Omron CX-Programmer project NewProject (CX-Programmer 9.73)

# PLC bagagli: CPM1(CPM1A) CPU20

## Global symbols (name address type ; comment)
0.01 BOOL  ; EntryBalance1
0.02 BOOL  ; SensorBalance2
0.03 BOOL  ; SensorBalance3
0.04 BOOL  ; WeightC1
0.05 BOOL  ; XRayC1
0.06 BOOL  ; WeightC2
0.07 BOOL  ; XRayC2
0.08 BOOL  ; WeightC3
0.09 BOOL  ; Tag3
0.10 BOOL  ; Tag
0.11 BOOL  ; SensorEntryRoll1
0.12 BOOL  ; SensorRoll2
0.13 BOOL  ; SensorRoll3
0.14 BOOL  ; SensorRoll2
0.15 BOOL  ; SensorRoll3
10.00 BOOL  ; BagOnBalance1
10.01 BOOL  ; Position Control1
10.02 BOOL  ; Position Control2
10.03 BOOL  ; Position Control3
10.04 BOOL  ; RemLW1
10.05 BOOL  ; RemLW2
10.06 BOOL  ; RemLW3
10.07 BOOL  ; Container brought to destination
10.08 BOOL  ; Roll3
10.09 BOOL  ; Roll2
10.10 BOOL  ; Roll1
10.11 BOOL  ; Roll1
10.12 BOOL  ; Roll2
10.13 BOOL  ; Roll3
10.14 BOOL  ; FlagCont
11.01 BOOL  ; Roll1
11.02 BOOL  ; Roll2
11.03 BOOL  ; Roll3
1.01 BOOL  ; EntryL1
1.02 BOOL  ; ExitL1
1.03 BOOL  ; EntryL2
1.04 BOOL  ; ExitL2
1.05 BOOL  ; EntryL3
1.06 BOOL  ; ExitL3
1.07 BOOL  ; Tag1
1.08 BOOL  ; Tag2
1.09 BOOL  ; Tag3
1.10 BOOL  ; Exit2Full
1.11 BOOL  ; EndRoll2
1.12 BOOL  ; ExitSensorRoll1
1.13 BOOL  ; SensorRoll3
1.14 BOOL  ; SensorRoll1
1.15 BOOL  ; SensorRoll2
CNT127 BOOL  ; ContainerL
HR0.01 BOOL  ; test1
HR0.04 BOOL  ; test1
TIM000 BOOL  ; 10s to change container

## Program NewProgram1 (no task)
Local symbols
SensorRoll2 1.15 BOOL  ; SensorRoll2
XRayC1 BOOL

### Section Section1

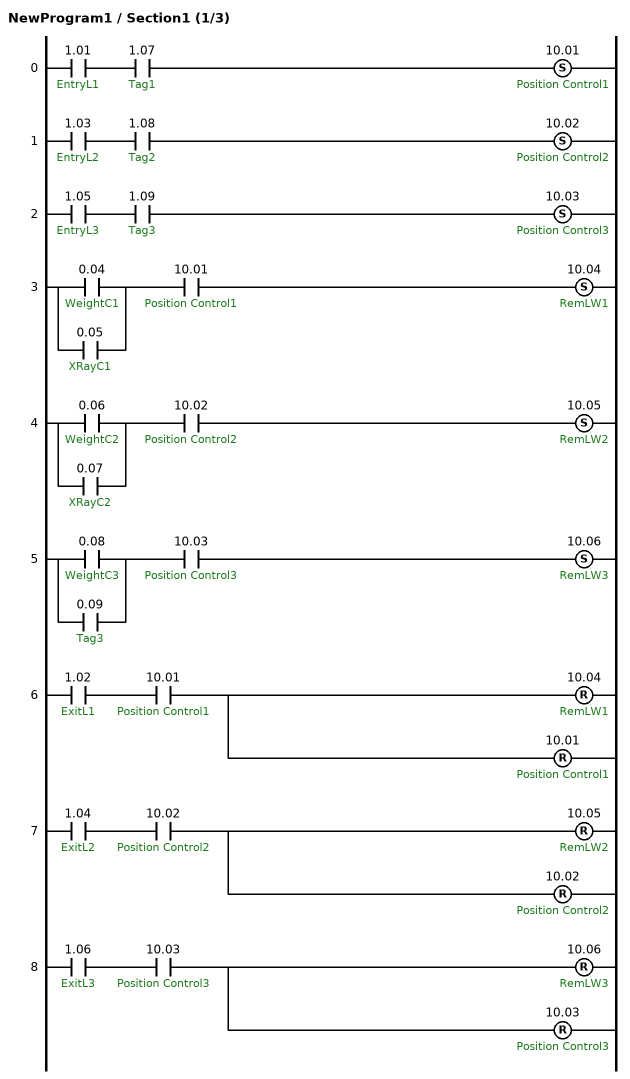
; rung 0
LD 1.01  ; EntryL1
AND 1.07  ; Tag1
SET 10.01  ; Position Control1
; rung 1
LD 1.03  ; EntryL2
AND 1.08  ; Tag2
SET 10.02  ; Position Control2
; rung 2
LD 1.05  ; EntryL3
AND 1.09  ; Tag3
SET 10.03  ; Position Control3
; rung 3
LD 0.04  ; WeightC1
OR 0.05  ; XRayC1
AND 10.01  ; Position Control1
SET 10.04  ; RemLW1
; rung 4
LD 0.06  ; WeightC2
OR 0.07  ; XRayC2
AND 10.02  ; Position Control2
SET 10.05  ; RemLW2
; rung 5
LD 0.08  ; WeightC3
OR 0.09  ; Tag3
AND 10.03  ; Position Control3
SET 10.06  ; RemLW3
; rung 6
LD 1.02  ; ExitL1
AND 10.01  ; Position Control1
RSET 10.04  ; RemLW1
RSET 10.01  ; Position Control1
; rung 7
LD 1.04  ; ExitL2
AND 10.02  ; Position Control2
RSET 10.05  ; RemLW2
RSET 10.02  ; Position Control2
; rung 8
LD 1.06  ; ExitL3
AND 10.03  ; Position Control3
RSET 10.06  ; RemLW3
RSET 10.03  ; Position Control3

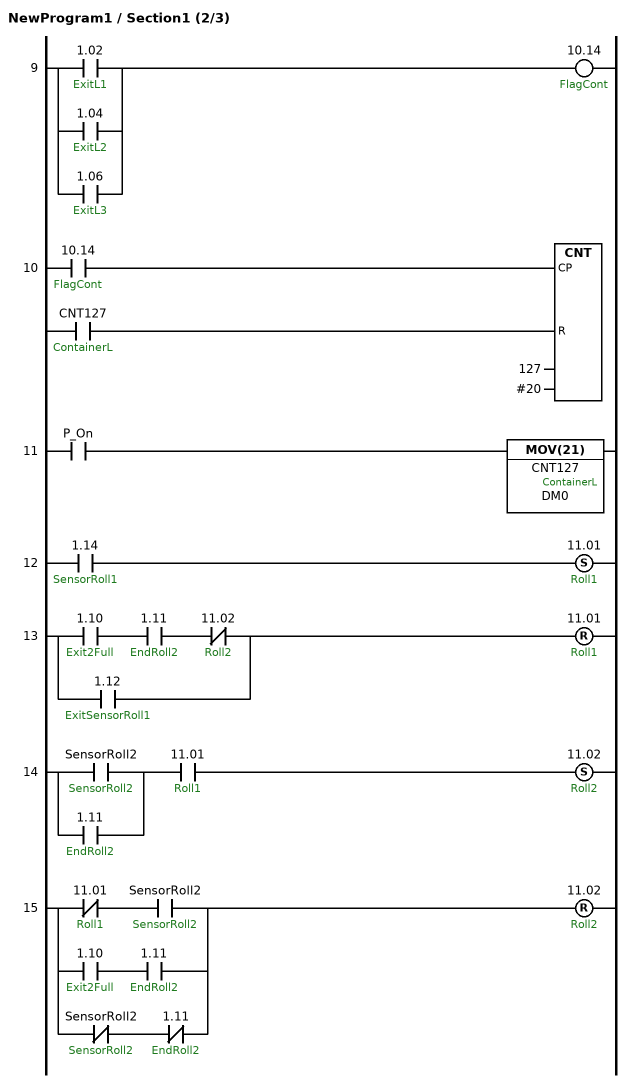
; rung 9
LD 1.02  ; ExitL1
OR 1.04  ; ExitL2
OR 1.06  ; ExitL3
OUT 10.14  ; FlagCont
; rung 10
LD 10.14  ; FlagCont
LD CNT127  ; ContainerL
CNT 127 #20
; rung 11
LD P_On
MOV(21) CNT127 DM0  ; ContainerL
; rung 12
LD 1.14  ; SensorRoll1
SET 11.01  ; Roll1
; rung 13
LD 1.10  ; Exit2Full
AND 1.11  ; EndRoll2
ANDNOT 11.02  ; Roll2
OR 1.12  ; ExitSensorRoll1
RSET 11.01  ; Roll1
; rung 14
LD SensorRoll2  ; SensorRoll2
OR 1.11  ; EndRoll2
AND 11.01  ; Roll1
SET 11.02  ; Roll2
; rung 15
LDNOT 11.01  ; Roll1
AND SensorRoll2  ; SensorRoll2
LD 1.10  ; Exit2Full
AND 1.11  ; EndRoll2
ORLD
LDNOT SensorRoll2  ; SensorRoll2
ANDNOT 1.11  ; EndRoll2
ORLD
RSET 11.02  ; Roll2

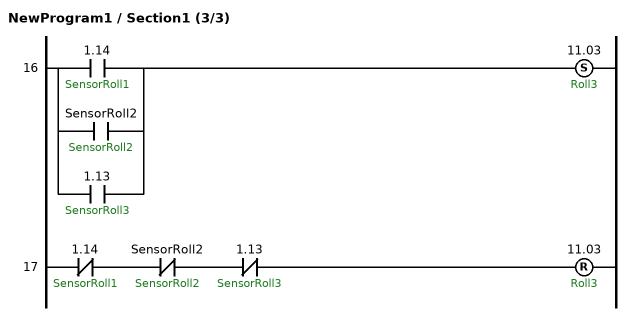
; rung 16
LD 1.14  ; SensorRoll1
OR SensorRoll2  ; SensorRoll2
OR 1.13  ; SensorRoll3
SET 11.03  ; Roll3
; rung 17
LDNOT 1.14  ; SensorRoll1
ANDNOT SensorRoll2  ; SensorRoll2
ANDNOT 1.13  ; SensorRoll3
RSET 11.03  ; Roll3

### Section END
; rung 0
END(01)